Yaskawa INFORM job: LOAD_TOP_START_XYZ.JBI

/JOB
//NAME LOAD_TOP_START_XYZ
///FOLDERNAME FOLDER001
//POS
///NPOS 0,0,0,1,0,0
///TOOL 1
///POSTYPE ROBOT
///RECTAN
///RCONF 1,0,0,0,0,0,0,0,0,0,0,0,0,0,0,0,0,0,0,0,0,0,0,0
P00124=792.896,161.791,493.972,179.9986,-9.9993,0.0008
//INST
///DATE 2025/09/26 17:00
///ATTR SC,RW
///GROUP1 RB1
NOP
'GET X Y Z VALUE FOR BOTTOM START
'X
GETE D061 P124 (1)
SET I061  EXPRESS I060 * 100
IFTHENEXP I061>10000
	 SET I061 10000
ELSEIFEXP I061<-10000
	 SET I061 -10000
ENDIF
'Y
GETE D063 P124 (2)
SET I063  EXPRESS I062 * 100
IFTHENEXP I063>10000
	 SET I063 10000
ELSEIFEXP I063<-10000
	 SET I063 -10000
ENDIF
'Z
GETE D065 P124 (3)
SET I065  EXPRESS I064 * 100
IFTHENEXP I065>10000
	 SET I065 10000
ELSEIFEXP I065<-10000
	 SET I065 -10000
ENDIF
'ADD THE CORRECTIONS
ADD D061 I061
SETE P124 (1) D061
ADD D063 I063
SETE P124 (2) D063
ADD D065 I065
SETE P124 (3) D065
'SET TO 0
SET I060 0
SET I061 0
SET I062 0
SET I063 0
SET I064 0
SET I065 0
END
